FUNCTION_BLOCK OnStackChangedHandler EXTENDS OnStackEventHandler

METHOD PUBLIC HandleEvent
VAR_INPUT
	Event : I_Event;
END_VAR
VAR
	stackChangedEvent : I_StackChangedEvent;
END_VAR
IF __QUERYINTERFACE(Event, stackChangedEvent) THEN
	_eventReceived := TRUE;
	fromExpected := stackChangedEvent.TargetStack = expectedOriginator;
END_IF
END_METHOD

END_FUNCTION_BLOCK

(* stored: Version 1.1.0.1, ProductVersion 3.1.4024.12
   POU OnStackChangedHandler: Id {b89d0093-c16c-4457-a9cc-9b4405520d6c}, SpecialFunc None
   Method HandleEvent: Id {3e8d5506-8c11-4b97-bd07-53573c6df22c} *)
